Staubli VAL3: Day5.pjx

--- Day5.pjx ---
Parameters version=s8.13.1Cs9_BS2800 stackSize=5000 millimeterUnit=true
Program file=get_int_points.pgx
Program file=size_grid.pgx
Program file=start.pgx
Program file=stop.pgx
Data file=Day5.dtx
Library alias=util path=Disk://helpers/helpers.pjx
Library alias=str path=Disk://string/string.pjx
Type name=lists path=Disk://types/lists/lists.pjx
Type name=lists_num path=Disk://types/lists_num/lists_num.pjx

--- Day5.dtx ---
string sInput
lists lResult
  [0]
    string sString
num nGrid[1 1]
lists lTemp
  [0]
    string sString
num nX1
num nY1
num nX2
num nY2
string sX1
string sY1
string sX2
string sY2
num nResRangeX
num nResRangeY
num nIntX
num nIntY

--- start.pgx ---
program start()
  local num l_nElement
  local num l_nCounter
  local string l_sLine
  local num l_nString
  local num l_nIntPoints
  local num l_nX
  local num l_nY
begin

  // read file
  call util:readFile("Disk://input_day5.txt", sInput)
  // sInput[0] = "905,103 -> 905,82"

  call str:splitString(sInput," -> ", lResult)

  resize(sX1, 1, size(lResult))
  resize(sY1, 1, size(lResult))
  resize(sX2, 1, size(lResult))
  resize(sY2, 1, size(lResult))

  // parse x1,y1,x2,y2 to string variables
  for l_nElement = 0 to size(lResult)-1
    for l_nString = 0 to size(lResult[l_nElement].sString)-1
      l_sLine = lResult[l_nElement].sString[l_nString]

      call str:splitString(l_sLine, ",", lTemp)
      if l_nString == 0
        sX1[l_nElement] = lTemp.sString[0]
        sY1[l_nElement] = lTemp.sString[1]
      else
        sX2[l_nElement] = lTemp.sString[0]
        sY2[l_nElement] = lTemp.sString[1]
      endIf
    endFor
  endFor

  // convert strings to nums
  call util:vec2num(sX1, nX1)
  call util:vec2num(sY1, nY1)
  call util:vec2num(sX2, nX2)
  call util:vec2num(sY2, nY2)

  call size_grid()

  // PUZZLE 1
  for l_nElement = 0 to size(nX1)-1
    call get_int_points(nX1[l_nElement],nY1[l_nElement],nX2[l_nElement],nY2[l_nElement], nIntX, nIntY)
    if((nX2[l_nElement]-nX1[l_nElement]) == 0) or ((nY2[l_nElement]-nY1[l_nElement]) == 0)
      for l_nIntPoints = 0 to min(size(nIntX), size(nIntY))-1
        nGrid[nIntX[l_nIntPoints],nIntY[l_nIntPoints]] = nGrid[nIntX[l_nIntPoints],nIntY[l_nIntPoints]] + 1
      endFor
    endIf
  endFor

  // now find entries in nGrid >=2
  l_nCounter = 0
  for l_nX = 0 to size(nGrid,1)-1
    for l_nY = 0 to size(nGrid,2)-1
      if nGrid[l_nX, l_nY] >=2
        l_nCounter = l_nCounter +1
      endIf
    endFor
  endFor

  call util:printNum(l_nCounter)
  // 6267


  // PUZZLE 2
 call size_grid()

  // start calculation
  for l_nElement = 0 to size(nX1)-1
    call get_int_points(nX1[l_nElement],nY1[l_nElement],nX2[l_nElement],nY2[l_nElement], nIntX, nIntY)
    for l_nIntPoints = 0 to min(size(nIntX), size(nIntY))-1
      nGrid[nIntX[l_nIntPoints],nIntY[l_nIntPoints]] = nGrid[nIntX[l_nIntPoints],nIntY[l_nIntPoints]] + 1
    endFor
  endFor

  // now find entries in nGrid >=2
  l_nCounter = 0
  for l_nX = 0 to size(nGrid,1)-1
    for l_nY = 0 to size(nGrid,2)-1
      if nGrid[l_nX, l_nY] >=2
        l_nCounter = l_nCounter +1
      endIf
    endFor
  endFor

  call util:printNum(l_nCounter)
  // 20196


end

--- get_int_points.pgx ---
program get_int_points(num x_nX1, num x_nY1, num x_nX2, num x_nY2, num& x_nResX[], num& x_nResY[])
  local num l_nElement
  local num l_nResLength[2]
  local num l_nSign[2]
begin

  resize(nResRangeX,1,1)
  nResRangeX = 0
  resize(nResRangeY,1,1)
  nResRangeY = 0

  resize(x_nResX,1,1)
  x_nResX = 0
  resize(x_nResY,1,1)
  x_nResY = 0

  l_nSign[0] = sel(x_nX1 > x_nX2, -1,1)
  l_nSign[1] = sel(x_nY1 > x_nY2, -1,1)

  if(x_nX1 - x_nX2) == 0 and (x_nY1 - x_nY2) != 0
    nResRangeX = x_nX1
    call util:range(x_nY1,x_nY2+1, l_nSign[1], nResRangeY)
  elseIf(x_nY1 - x_nY2) == 0 and (x_nX1 - x_nX2) != 0
    call util:range(x_nX1,x_nX2+1, l_nSign[0], nResRangeX)
    nResRangeY = x_nY1
  elseIf(x_nX1 - x_nX2) == 0 and (x_nY1 - x_nY2) == 0
    nResRangeX = x_nX1
    nResRangeY = x_nY1
  else
    call util:range(x_nX1,x_nX2+1, l_nSign, nResRangeX)
    call util:range(x_nY1,x_nY2+1, l_nSign[1], nResRangeY)
  endIf

  l_nResLength[0] = max(size(nResRangeX), size(nResRangeY))
  l_nResLength[1] = min(size(nResRangeX), size(nResRangeY))

  resize(x_nResX,1,1)
  x_nResX = 0
  resize(x_nResX,1,l_nResLength)
  resize(x_nResY,1,1)
  x_nResY = 0
  resize(x_nResY,1,l_nResLength)

  if size(nResRangeX) == size(nResRangeY)
    // diagonals
    for l_nElement = 0 to l_nResLength[0]-1
      x_nResX[l_nElement] = nResRangeX[l_nElement]
      x_nResY[l_nElement] = nResRangeY[l_nElement]
    endFor
  else
    // horizontal or vertical
    for l_nElement = 0 to l_nResLength[0]-1
      if size(nResRangeX) == 1
        // x-coordinate is not changing -> keep constant
        x_nResX[l_nElement] = nResRangeX
        x_nResY[l_nElement] = nResRangeY[l_nElement]
      else
        x_nResX[l_nElement] = nResRangeX[l_nElement]
        x_nResY[l_nElement] = nResRangeY
      endIf

    endFor

  endIf

end

--- size_grid.pgx ---
program size_grid()
  local num l_nGridMax[2]
begin

  // helpers
  resize(nGrid,1,1)
  resize(nGrid,2,1)
  nGrid[0,0]=0

  // size grid
  call util:vecMax(nX1, l_nGridMax[0])
  call util:vecMax(nX2, l_nGridMax[1])
  resize(nGrid,1,max(l_nGridMax[0], l_nGridMax[1])+1)

  call util:vecMax(nY1, l_nGridMax[0])
  call util:vecMax(nY2, l_nGridMax[1])
  resize(nGrid,2,max(l_nGridMax[0], l_nGridMax[1])+1)
end
